TYPE MyCustomType :
STRUCT
    isActive : BOOL;
    speed    : REAL;
    counter  : INT;
END_STRUCT
END_TYPE

(* stored: Version 1.1.0.1, ProductVersion 3.1.4024.15
   DUT MyCustomType: Id {32b183df-521f-409a-ac06-dc747254f394} *)
